{attribute addProperty BoxType "EK1100-0000-0018"}
{attribute addProperty Id "Beckhoff_ATH2xxxEK1122Beckhoff_ATH2xxxEK1122_63628BEE6960870A_0013_ATH2000_5250_0022ATH2000_490CE0DD11214"}
{attribute addProperty CRC "1210179214"}
{attribute addProperty SizeInBites "7072"}
{attribute addProperty SizeInBytes "884"}
TYPE Beckhoff_ATH2xxx_4821DE8E EXTENDS EK1100_179A0949 :
STRUCT
	{attribute addProperty Name "Beckhoff_ATH2xxxEK1122"}
	Beckhoff_ATH2xxxEK1122 : Beckhoff_ATH2xxxEK1122_63628BEE;
	{attribute addProperty Name "A_0013_ATH2000_5250_0022"}
	A_0013_ATH2000_5250_0022 : ATH2000_490CE0DD;
END_STRUCT
END_TYPE

(* stored: Version 1.2.0.0, ProductVersion 3.1.4024.9
   DUT Beckhoff_ATH2xxx_4821DE8E: Id {0475225a-d073-4120-aed3-1ee096172cfa} *)
